FUNCTION_BLOCK L3_PartRouterT (* Part Router based on part type *)
  (* Standard: 61499-2 *)
  (* Version 0.0, 2014-09-24, EQUEROL, UJI *)
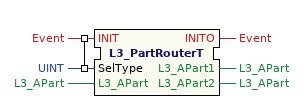
  EVENT_INPUT
    INIT WITH SelType; (* Initialization Request *)
  END_EVENT
  EVENT_OUTPUT
    INITO; (* Initialization Confirm *)
  END_EVENT
  VAR_INPUT
    SelType : UINT; (* Routing condition *)
  END_VAR
  SOCKETS
    L3_APart : L3_APart; (* Input Part *)
  END_SOCKETS
  PLUGS
    L3_APart1 : L3_APart; (* Output Part 1 *)
    L3_APart2 : L3_APart; (* Output part 2 *)
  END_PLUGS
  VAR
    Select : BOOL := FALSE; (* Variable to select output event *)
  END_VAR
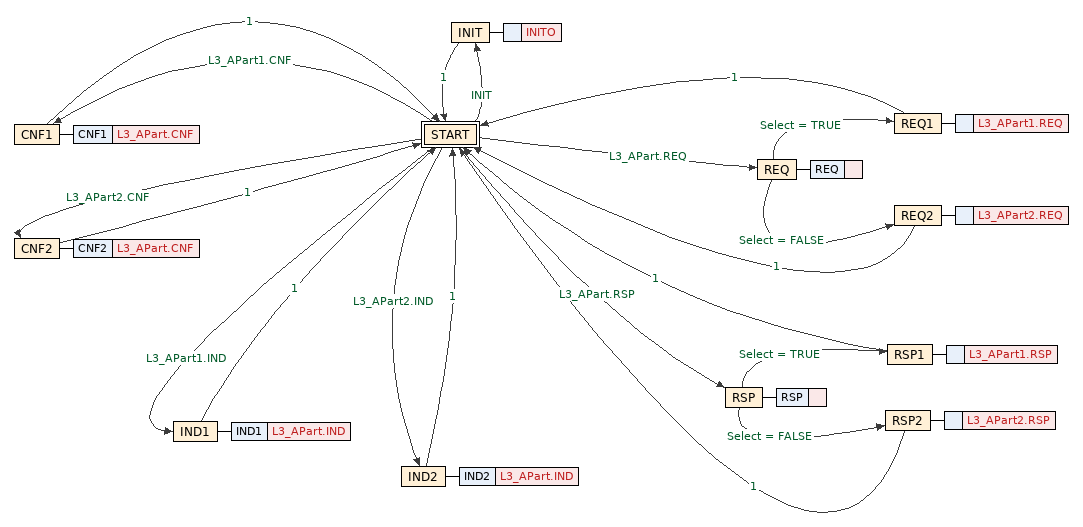
  EC_STATES
    START; (* Initial State *)
    INIT : -> INITO; (* Initialization *)
    REQ : REQ;
    REQ1 : -> L3_APart1.REQ;
    REQ2 : -> L3_APart2.REQ;
    RSP : RSP;
    RSP1 : -> L3_APart1.RSP;
    RSP2 : -> L3_APart2.RSP;
    CNF1 : CNF1 -> L3_APart.CNF;
    IND1 : IND1 -> L3_APart.IND;
    CNF2 : CNF2 -> L3_APart.CNF;
    IND2 : IND2 -> L3_APart.IND;
  END_STATES
  EC_TRANSITIONS
    START TO INIT := INIT;
    INIT TO START := 1;
    START TO REQ := L3_APart.REQ;
    REQ TO REQ1 := Select = TRUE;
    REQ TO REQ2 := Select = FALSE;
    REQ1 TO START := 1;
    REQ2 TO START := 1;
    START TO RSP := L3_APart.RSP;
    RSP TO RSP1 := Select = TRUE;
    RSP TO RSP2 := Select = FALSE;
    RSP1 TO START := 1;
    RSP2 TO START := 1;
    START TO CNF1 := L3_APart1.CNF;
    CNF1 TO START := 1;
    START TO IND1 := L3_APart1.IND;
    IND1 TO START := 1;
    START TO CNF2 := L3_APart2.CNF;
    CNF2 TO START := 1;
    START TO IND2 := L3_APart2.IND;
    IND2 TO START := 1;
  END_TRANSITIONS
  ALGORITHM REQ IN ST: (* Routes REQ event and data *)
IF L3_APart.TypeP = SelType THEN
(*Map input request to output 1*)
L3_APart1.PartIDP := L3_APart.PartIDP;
L3_APart1.FamilyP := L3_APart.FamilyP;
L3_APart1.TypeP := L3_APart.TypeP;
L3_APart1.Lotsize := L3_APart.Lotsize;
L3_APart1.Deadline := L3_APart.Deadline;
Select := TRUE;

ELSE
(*Map input request to output 2*)
L3_APart2.PartIDP := L3_APart.PartIDP;
L3_APart2.FamilyP := L3_APart.FamilyP;
L3_APart2.TypeP := L3_APart.TypeP;
L3_APart2.Lotsize := L3_APart.Lotsize;
L3_APart2.Deadline := L3_APart.Deadline;
Select := FALSE;

END_IF;
  END_ALGORITHM
  ALGORITHM RSP IN ST: (* Routes RSP event and data *)
IF L3_APart.TypeP = SelType THEN
(*Map input request to output 1*)
L3_APart1.FamilyP := L3_APart.FamilyP;
L3_APart1.TypeP := L3_APart.TypeP;
L3_APart1.Deadline := L3_APart.Deadline;
Select := TRUE;

ELSE
(*Map input request to output 2*)
L3_APart2.FamilyP := L3_APart.FamilyP;
L3_APart2.TypeP := L3_APart.TypeP;
L3_APart2.Deadline := L3_APart.Deadline;
Select := FALSE;

END_IF;
  END_ALGORITHM
  ALGORITHM CNF1 IN ST: (* Routes CNF1 event and data *)
(*No data needs to be mapped in this case*)
(*To be used in the future if is needed to return any data with CNF event*)
  END_ALGORITHM
  ALGORITHM IND1 IN ST: (* Routes IND1 event and data *)
(*Map input IND1 to common output*)
L3_APart.PartIDS := L3_APart1.PartIDS;
L3_APart.FamilyS := L3_APart1.FamilyS;
L3_APart.TypeS := L3_APart1.TypeS;
  END_ALGORITHM
  ALGORITHM CNF2 IN ST: (* Routes CNF2 event and data *)
(*No data needs to be mapped in this case*)
(*To be used in the future if is needed to return any data with CNF event*)
  END_ALGORITHM
  ALGORITHM IND2 IN ST: (* Routes IND2 event and data *)
(*Map input IND2 to common output*)
L3_APart.PartIDS := L3_APart2.PartIDS;
L3_APart.FamilyS := L3_APart2.FamilyS;
L3_APart.TypeS := L3_APart2.TypeS;
  END_ALGORITHM
END_FUNCTION_BLOCK
